# EPICS substitutions: bpmApp/Db/fofb.substitutions
#
#
#	MSGID   : Waveform Message ID
#	PID		: Power Supply ID
#	KP		: Kp Memory address
#	KI		: Ki Memory Address
#	KD		: Kd Memory Address
#
file fofb.template
{ pattern
	{P,     MSGID, PID, ID_ADDR, KP, KI, KD, LEN, A1, A2, A3, A4, A5, A6 }
	{ "\$(P)", 74, 1,   560, 800, 848, 896, 540, 160, 208,608, 800, 848, 896 }
	{ "\$(P)", 75, 2,   564, 804, 852, 890, 540, 164, 212,612, 804, 852, 900  }
	{ "\$(P)", 76, 3,   568, 808, 856, 894, 540, 168, 216,616, 808, 856, 904  }
	{ "\$(P)", 77, 4,   572, 812, 860, 898, 540, 172, 220,620, 812, 860, 908  }
	{ "\$(P)", 78, 5,   576, 816, 864, 902, 540, 176, 224,624, 816, 864, 912  }
	{ "\$(P)", 79, 6,   580, 820, 868, 906, 540, 180, 228,628, 820, 868, 916  }
	{ "\$(P)", 80, 7,   584, 824, 872, 910, 540, 184, 232,632, 824, 872, 920  }
	{ "\$(P)", 81, 8,   592, 828, 876, 914, 540, 188, 236,636, 828, 876, 924  }
	{ "\$(P)", 82, 9,   596, 832, 880, 918, 540, 192, 240,640, 832, 880, 928  }
	{ "\$(P)", 83, 10,  600, 836, 884, 922, 540, 196, 244,644, 836, 884, 932  }
	{ "\$(P)", 84, 11,  604, 840, 888, 926, 540, 200, 248,648, 840, 888, 936  }
	{ "\$(P)", 85, 12,  608, 844, 892, 930, 540, 204, 252,652, 844, 892, 940  }
}
